{attribute 'qualified_only'}
TYPE E_LevelSelector : (
	
    eUpperOnly := 1,   // Only upper level enabled
    eLowerOnly := 2,   // Only lower level enabled
    eBoth      := 3    // Upper + Lower enabled
);
END_TYPE

(* stored: Version 1.1.0.1
   DUT E_LevelSelector: Id {1b042426-21a5-4cd1-ac46-1d49e42fca74} *)
